PROGRAM P_DeadBand
VAR
	fbDeadBandOne : FB_DeadBand;
	fbDeadBandTwo : FB_DeadBand;
END_VAR

fbDeadBandOne(
	fSignal := 0.0,
	fDeadBandUp := G_Parameters.fDeadUpOne,
	fDeadBanddown := G_Parameters.fDeadDownOne,
	fXDotRef := G_Parameters.fMaxSpeedMain * G_OPC.fJoystickMain,
	fCompansatedSignal =>G_OPC.fValveOneCompansatedOut
);

fbDeadBandTwo(
	fSignal := 0.0,
	fDeadBandUp := G_Parameters.fDeadUpTwo,
	fDeadBanddown := G_Parameters.fDeadDownTwo,
	fXDotRef := G_Parameters.fMaxSpeedJib * G_OPC.fJoystickJib,
	fCompansatedSignal =>G_OPC.fValveTwoCompansatedOut
);

END_PROGRAM

(* stored: Version 1.1.0.1
   POU P_DeadBand: Id {492067f6-deee-408c-a414-4c49d135cc0d}, SpecialFunc None *)
